(* IEC 61131-3 sources: CodesysTest/export/Testing/Motors/Applied Motion, 7 files *)

(* ---- eAppliedMotionDriveStates.dut.st ---- *)
(*#-#-#-#-#-#-#-#-#-#---Declaration---#-#-#-#-#-#-#-#-#-#-#-#-#*)

{attribute 'qualified_only'}
{attribute 'strict'}
TYPE eAppliedMotionDriveStates :
(
	Idle := 0,
	MoveABS := 10,
	MovePush := 11,
	MoveInc := 12,
	SendPars := 40,
	SendOpcodeAfterPars := 41,
	Jogging := 20,
	Moving := 50,
	DoneMoving := 51,
	Halt := 60,
	Halting := 61,
	Halted := 62,
	Home := 70,
	Homing := 71,
	Faulting := 98,
	Faulted := 99
);
END_TYPE

(* ---- eAppliedMotionDriveStatesASCII.dut.st ---- *)
(*#-#-#-#-#-#-#-#-#-#---Declaration---#-#-#-#-#-#-#-#-#-#-#-#-#*)

{attribute 'qualified_only'}
{attribute 'strict'}
TYPE eAppliedMotionDriveStatesASCII :
(
	Idle := 0,
	MoveABS := 10,
	MovePush := 11,
	MoveInc := 12,
	SendPars := 40,
	SendOpcodeAfterPars := 41,
	Jogging := 20,
	Moving := 50,
	DoneMoving := 51,
	Halt := 60,
	Halting := 61,
	Halted := 62,
	Home := 70,
	Homing := 71,
	Faulting := 98,
	Faulted := 99
);
END_TYPE

(* ---- eAppliedMotionOpcodes.enum.st ---- *)
(*#-#-#-#-#-#-#-#-#-#---Declaration---#-#-#-#-#-#-#-#-#-#-#-#-#*)

{attribute 'strict'}
{attribute 'qualified_only'}
//Taken from Host-Command-Reference pdf on Applied Motion website
TYPE eAppliedMotionOpcodes :
(
	ALARM_RESET := 16#BA,
	START_JOGGING := 16#96,
	STOP_JOGGING := 16#D8,
	ENCODER_FUNCTION := 16#D6,     //0
	ENCODER_POSITION := 16#98,     //Position
	FEED_TO_DOUBLE_SENSOR := 16#69,     //I/O Point 1 Condition 1 I/O Point 2 Condition 2
	FOLLOW_ENCODER := 16#CC,     //I/O Point Condition
	FEED_TO_LENGTH := 16#66,
	FEED_TO_SENSOR_WITH_MASK_DISTANCE := 16#6A,     //I/O Point Condition
	FEED_AND_SET_OUTPUT := 16#68,     //I/O Point Condition
	FEED_TO_POSITION := 16#67,
	FEED_TO_SENSOR := 16#6B,     //I/O Point Condition
	FEED_TO_SENSOR_WITH_SAFETY_DISTANCE := 16#6C,     //I/O Point Condition
	JOG_DISABLE := 16#A3,
	JOG_ENABLE := 16#A2,
	MOTOR_DISABLE := 16#9E,
	MOTOR_ENABLE := 16#9F,
	SEEK_HOME := 16#6E,     //I/O Point Condition
	SET_POSITION := 16#A5,     //Position
	FILTER_INPUT := 16#C0,     //I/O Point Filter Time
	FILTER_SELECT_INPUTS := 16#D3,
	STEP_FILTER_FREQ := 16#06,     //Freq
	ANALOG_DEADBAND := 16#D2,     //0.001 V
	ALARM_RESET_INPUT := 16#46,     //Function ('1'..'3') I/O Point
	ALARM_OUTPUT := 16#47,     //Function ('1'..'3') I/O Point
	ANALOG_SCALING := 16#D1,
	DEFINE_LIMITS := 16#42,     //1..3
	SET_OUTPUT := 16#8B,     //I/O Point Condition
	WAIT_FOR_INPUT := 16#70,
	QUEUE_LOAD_AND_EXECUTE := 16#78,     //1..12
	WAIT_TIME := 16#6F,     //0.01 sec
	STOP_MOVE_KILL_BUFFER := 16#E1,
	STOP_MOVE_KILL_BUFFER_NORMAL_DECEL := 16#E2,
	STOP_MOVE := 16#B5  // Might work, might not
);
END_TYPE

(* ---- eOrientalOperationType_1.dut.st ---- *)
(*#-#-#-#-#-#-#-#-#-#---Declaration---#-#-#-#-#-#-#-#-#-#-#-#-#*)

{attribute 'qualified_only'}
{attribute 'strict'}
TYPE eOrientalOperationType_1 :
(
	No_Setting := 0,
	Absolute_Positioning := 1,
	Incremental_Positioning := 2,
	Absolute_Push := 20,
	Incremental_Push := 21
);
END_TYPE

(* ---- sctAppliedMotionPars.dut.st ---- *)
(*#-#-#-#-#-#-#-#-#-#---Declaration---#-#-#-#-#-#-#-#-#-#-#-#-#*)

TYPE sctAppliedMotionPars :
STRUCT
	Position : uModbusDWORD;
	Speed : WORD;
	Accel : WORD;
	Decel : WORD;
END_STRUCT
END_TYPE

(* ---- FB_AppliedMotionAlarms.pou.st ---- *)
(*#-#-#-#-#-#-#-#-#-#---Declaration---#-#-#-#-#-#-#-#-#-#-#-#-#*)

FUNCTION_BLOCK FB_AppliedMotionAlarms
VAR_INPUT
    alarmCode : WORD;
END_VAR
VAR_OUTPUT
    positionLimit : BOOL;        // FAULT - Motor exceeded position limit - following error
    CCWLimit : BOOL;      // WARNING - Motor is at CCW Limit
    CWLimit : BOOL;      // WARNING - Motor is at CW Limit
    overTemp : BOOL;      // FAULT - Motor Over Temperature Limit
    internalVoltage : BOOL;      // FAULT - Internal Voltage Fault
    overVoltage : BOOL;      // FAULT - Overvoltage Fault
    underVoltage : BOOL;      // WARNING - Undervoltage Warning
    overCurrent : BOOL;      // FAULT - Motor Overcurrent
    openMotorWinding : BOOL;      // FAULT - Motor Detected Open Winding
    badEncoder : BOOL;      // FAULT - Motor Encoder Failure
    commError : BOOL;      // WARNING - Communications Error
    badFlash : BOOL;      // WARNING - Bad Flash
    noMove : BOOL;      // WARNING - No Move
    currentFoldback  : BOOL;      // WARNING - Current Foldback
    blankQSegment : BOOL;      // WARNING - Blank Q Segment
    NVMemoryDoubleError : BOOL;      // WARNING - NV Memory Double Error
END_VAR
VAR
END_VAR
(*#-#-#-#-#-#-#-#-#-#---Implementation---#-#-#-#-#-#-#-#-#-#-#-#-#*)

//    Fucntion Block: FB_StepServoAlarms
//    Description: This unpacks the step servo alarm bits from the alarm word received over EIP
//    Created by: Ben Hess
//    Created Date: September 5th, 2018

positionLimit := alarmCode.0;
CCWLimit := alarmCode.1;
CWLimit := alarmCode.2;
overTemp := alarmCode.3;
internalVoltage := alarmCode.4;
overVoltage := alarmCode.5;
underVoltage := alarmCode.6;
overCurrent    := alarmCode.7;
openMotorWinding := alarmCode.8;
badEncoder := alarmCode.9;
commError := alarmCode.10;
badFlash := alarmCode.11;
noMove := alarmCode.12;
currentFoldback := alarmCode.13;
blankQSegment := alarmCode.14;
NVMemoryDoubleError := alarmCode.15;

(* ---- FB_AppliedMotionStatus.pou.st ---- *)
(*#-#-#-#-#-#-#-#-#-#---Declaration---#-#-#-#-#-#-#-#-#-#-#-#-#*)

FUNCTION_BLOCK FB_AppliedMotionStatus
VAR_INPUT
	statusCode : WORD;
END_VAR
VAR_OUTPUT
	motorEnabled : BOOL;		//Motor Enabled (Motor Disabled if this bit = 0)
	sampling : BOOL; 	 //Sampling (for Quick Tuner)
	driveFaulted : BOOL; 	 //Drive Fault (check Alarm Code)
	inPosition : BOOL; 	 //In Position (motor is in position)
	moving : BOOL; 	 //Moving (motor is moving)
	jogging	: BOOL; 	 //Jogging (currently in jog mode)
	stopping : BOOL; 	 //Stopping (in the process of stopping from a stop command)
	waitingForInput : BOOL; 	 //Waiting (for an input; executing a WI command)
	saving : BOOL; 	 //Saving (parameter data is being saved)
	alarmPresent : BOOL; 	 //Alarm present (check Alarm Code)
	homing : BOOL; 	 //Homing (executing an SH command)
	waitingForTime : BOOL; 	 //Waiting (for time; executing a WD or WT command)
	wizardRunning : BOOL; 	 //Wizard running (Timing Wizard is running)
	checkingEncoder	: BOOL; 	 //Checking encoder (Timing Wizard is running)
	Q_ProgramRunning : BOOL; 	 //Q Program is running
	initializing : BOOL; 	 //Initializing (happens at power up) ; Servo Ready (for SV200 drives only)
END_VAR
VAR
END_VAR
(*#-#-#-#-#-#-#-#-#-#---Implementation---#-#-#-#-#-#-#-#-#-#-#-#-#*)

//	Fucntion Block: StepServoStatus
//	Description: This unpacks the step servo status bits from the status word received over modbus
//	Created by: Ben Hess
//	Created Date: January 26th, 2018

motorEnabled := statusCode.0;
sampling := statusCode.1;
driveFaulted := statusCode.2;
inPosition := statusCode.3;
moving := statusCode.4;
jogging := statusCode.5;
stopping := statusCode.6;
waitingForInput	:= statusCode.7;
saving := statusCode.8;
alarmPresent := statusCode.9;
homing := statusCode.10;
waitingForTime := statusCode.11;
wizardRunning := statusCode.12;
checkingEncoder := statusCode.13;
Q_ProgramRunning := statusCode.14;
initializing := statusCode.15;
